// Mitsubishi GX Works2 project: b02   PLC: Q02/Q02H

PROGRAM MAIN
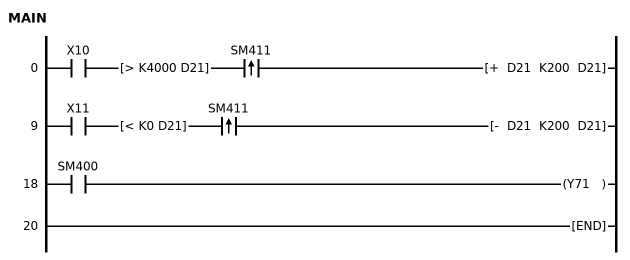
0     LD      X10
      AND>    K4000 D21
      ANDP    SM411
      +       D21 K200 D21
9     LD      X11
      AND<    K0 D21
      ANDP    SM411
      -       D21 K200 D21
18    LD      SM400
      OUT     Y71
20    END
END_PROGRAM
